// TIA Portal project "GaraznaVrata" (V17)

(* hardware
DEVICE "S7-1200 station_1"  S7-1200 Station
   slot 0: "Rack_0"  S7-1200 Rack  Rack  V1.0
   slot 1: "PLC_1"  CPU 1214C DC/DC/DC  6ES7 214-1AG40-0XB0  V4.2
DEVICE "HMI_1"  TP1200 Comfort
   slot 0: "HMI_1"  TP1200 Comfort  6AV2 124-0MC01-0AX0  17.0.0.0
   slot 1: "HMI_RT_1"  TP1200 Comfort  6AV2 124-0MC01-0AX0  17.0.0.0
   slot 5: "HMI_1.IE_CP_1"  PROFINET Interface  17.0.0.0
      slot 1: "PROFINET Interface_1"  PROFINET Interface
         slot 1: "Port_1"  Port
         slot 2: "Port_2"  Port
   slot 7: "HMI_1.MPI/DP_CP_1"  MPI/DP Interface  17.0.0.0
DEVICE "S7-1500/ET200MP station_1"  S7-1500 station
   slot 0: "Rail_0"  Rack  6ES7 590-1***0-0AA0
   slot 1: "PLC_2"  CPU 1513-1 PN  6ES7 513-1AL01-0AB0  V2.9
      slot 3: "CPU display_1"  6ES7591-1AA00-0AA0
      slot 32768: "PROFINET interface_1"  X1
         slot 32769: "Port_1"  X1 P1
         slot 32770: "Port_2"  X1 P2
      slot 34817: "Virtual CP interface port_1"  Virtual CP interface port  Virtual CP interface port
*)

// ===== PLC "PLC_1"  CPU 1214C DC/DC/DC =====

VAR_GLOBAL   // PLC tag table "Default tag table"
   "System_Byte" AT %MB1 : Byte;
   "FirstScan" AT %M1.0 : Bool;
   "DiagStatusUpdate" AT %M1.1 : Bool;
   "AlwaysTRUE" AT %M1.2 : Bool;
   "AlwaysFALSE" AT %M1.3 : Bool;
   "Clock_Byte" AT %MB0 : Byte;
   "Clock_10Hz" AT %M0.0 : Bool;
   "Clock_5Hz" AT %M0.1 : Bool;
   "Clock_2.5Hz" AT %M0.2 : Bool;
   "Clock_2Hz" AT %M0.3 : Bool;
   "Clock_1.25Hz" AT %M0.4 : Bool;
   "Clock_1Hz" AT %M0.5 : Bool;
   "Clock_0.625Hz" AT %M0.6 : Bool;
   "Clock_0.5Hz" AT %M0.7 : Bool;
END_VAR

VAR_GLOBAL   // PLC tag table "Tag table_1"
   "T1" AT %I0.0 : Bool;
   "T2" AT %I0.1 : Bool;
   "S1" AT %I0.2 : Bool;
   "KO" AT %I0.3 : Bool;
   "KZ" AT %I0.4 : Bool;
   "K1" AT %I0.5 : Bool;
   "K2" AT %I0.6 : Bool;
   "MZS" AT %I0.7 : Bool;
   "OTV" AT %Q0.0 : Bool;
   "ZAT" AT %Q0.1 : Bool;
   "ALM" AT %Q0.2 : Bool;
END_VAR

DATA_BLOCK "Block_2_DB"   // DB2
{ S7_Optimized_Access := 'TRUE' }
VERSION : 0.1
// stored: InstanceOfName Block_2
"Block_2"
BEGIN
END_DATA_BLOCK

FUNCTION_BLOCK "Block_2"   // FB1, SCL
{ S7_Optimized_Access := 'TRUE' }
VERSION : 0.1
   VAR_INPUT
      T1 : Bool;   // Inside push button
      T2 : Bool;   // Outside push button
      S1 : Bool;   // Inside comb switch
      KO : Bool;   // Signal "doors are open"
      KZ : Bool;   // Signal "doors are closed"
      K1 : Bool;   // Doors are opening
      K2 : Bool;   // Doors are closing
      MZS : Bool;   // Motor protection switch
   END_VAR
   VAR_OUTPUT
      OTV : Bool;   // Command to open the door
      ZAT : Bool;   // Command to close the door
      ALM : Bool;   // Alarm
   END_VAR
   VAR_IN_OUT
      M_BIT2 : Bool;   // temp bit for T2
      M_BIT : Bool;   // temp bit for T1
   END_VAR
   VAR
      sAlarm_MZS : Bool;   // Flag for MZS alarm
      sAlarm_KOKZ : Bool;   // Flag for KO and KZ alarm
      sAlarm_stuck : Bool;   // Flag for if gate didnt close/open
      sAlarm_K1K2 : Bool;   // Flag for K1 or K2 alarm
      sCls_gate : Bool;   // Flag to close the door
      sOpn_gate : Bool;   // Flag to open the door
      sGate_dir : Bool;   // Remember the last dirrection of the gate
      sOpening : Bool;   // temp var for opening gate
      sClosing : Bool;   // temp var for closing gate
      IEC_Timer_30s_alarm : TON_TIME;   // Timer for alarm_stuck
      IEC_Timer_5s_alarm : TON_TIME;   // Timer for alarm_K1K2
      IEC_Timer_2min_alarm : TON_TIME;   // Timer when door's are open
   END_VAR
   VAR_TEMP
      xPerm_opn : Bool;   // Permission to open the door
      xPerm_cls : Bool;   // Permission to close the door
      xT : Time;
      xAuto_close : Bool;   // Flag to auto close the door
   END_VAR
   VAR CONSTANT
      timer_2min : Time := T#2m;
      timer_5s : Time := T#5s;
      timer_30s : Time := T#30s;
   END_VAR
BEGIN
     REGION _AUTO_CLOSE
       // If gate is opened more than 2 min close it
       #IEC_Timer_2min_alarm(IN := #KO,
                             PT := #timer_2min,
                             Q => #xAuto_close,
                             ET => #xT);


       IF #xAuto_close THEN
           #sCls_gate := TRUE;
       END_IF;
   END_REGION

     REGION _PERMISSIONS
         // Permissions open the door
         IF #KZ AND NOT (#sAlarm_MZS OR #sAlarm_K1K2 OR #sAlarm_KOKZ OR #sAlarm_stuck) THEN
             #xPerm_opn := TRUE;
         ELSE
             #xPerm_opn := FALSE;
         END_IF;

         // Permission to close the door
         IF #KO AND NOT (#sAlarm_MZS OR #sAlarm_K1K2 OR #sAlarm_KOKZ OR #sAlarm_stuck) THEN
             #xPerm_cls := TRUE;
         ELSE
             #xPerm_cls := FALSE;
         END_IF;
     END_REGION

     REGION _PUSH_BUTTON_EVENT
         // T1 or T2 is pushed
         IF (#T1 AND NOT (#M_BIT)) XOR (#S1 AND (#T2 AND NOT (#M_BIT2))) THEN

             //open
             IF #xPerm_opn THEN
                 #sOpn_gate := TRUE;
             END_IF;

             //close
             IF #xPerm_cls THEN
                 #sCls_gate := TRUE;
             END_IF;

             //resume opening/closing door after error
             IF (#sAlarm_MZS OR #sAlarm_K1K2 OR #sAlarm_KOKZ OR #sAlarm_stuck) = FALSE AND #KO = FALSE AND #KZ = FALSE THEN
                 IF #sGate_dir THEN
                     #sOpn_gate := TRUE;
                 ELSE
                     #sCls_gate := TRUE;
                 END_IF;
             END_IF;

             // alarm shut down
             IF #sAlarm_MZS OR #sAlarm_K1K2 OR #sAlarm_KOKZ OR #sAlarm_stuck THEN
                 #sAlarm_MZS := FALSE;
                 #sAlarm_K1K2 := FALSE;
                 #sAlarm_KOKZ := FALSE;
                 #sAlarm_stuck := FALSE;
             END_IF;

             // set temp variables
             #sOpening := #sOpn_gate;
             #sClosing := #sCls_gate;

         END_IF;

         //set temp bit for edge detecting
         #M_BIT := #T1;
         #M_BIT2 := #T2;
     END_REGION

     REGION _REMEMBER_LAST_DIRRECTION
         // Remember the last direction
         IF #sOpn_gate THEN
             #sGate_dir := TRUE; // last dirrection of the gate was 'open'
         ELSIF #sCls_gate THEN
             #sGate_dir := FALSE; // last dirrection of the gate was 'close'
         END_IF;
     END_REGION

     REGION _OPEN/CLOSE_GATE
         // Start opening
         #OTV := #sOpn_gate;

         // Start Closing
         #ZAT := #sCls_gate;


         // Stop the opening
         IF #KO THEN
             #sOpn_gate := FALSE;
             #sOpening := #sOpn_gate;
         END_IF;

         // Stop the closing
         IF #KZ THEN
             #sCls_gate := FALSE;
             #sClosing := #sCls_gate;
         END_IF;
     END_REGION

     REGION _ALARMS


         (*
           alarm_MZS -> MZS error
           alarm_KOKZ -> Both KZ and K0 are active
           alarm_stuck -> If door didnt close or open within 30sec
           alarm_K1K2 -> Direction confirmation(K1 or K2) did not come within 5 sec of opening/closing gate
          *)

         //Send alarm signal
         IF #sAlarm_MZS OR #sAlarm_K1K2 OR #sAlarm_KOKZ OR #sAlarm_stuck THEN
             #sOpn_gate := FALSE;
             #sCls_gate := FALSE;
             #ALM := "Clock_0.5Hz";
         ELSE
             #ALM := FALSE;
         END_IF;

         //Direction confirmation did not come within 5 sec
         #IEC_Timer_5s_alarm(IN := ((#sOpening AND NOT #K1) OR (#sClosing AND NOT #K2)),
                             PT := #timer_5s,
                             Q => #sAlarm_K1K2,
                             ET => #xT);


         //If door didnt close or open within 30sec
         #IEC_Timer_30s_alarm(IN := #sOpening OR #sClosing,
                              PT := #timer_30s,
                              Q => #sAlarm_stuck,
                              ET => #xT);


         //MZS error
         IF #MZS THEN
             #sAlarm_MZS := TRUE;
         END_IF;

         //Both KZ and K0 are active
         IF #KZ AND #KO THEN
             #sAlarm_KOKZ := TRUE;
         END_IF;

     END_REGION
END_FUNCTION_BLOCK

ORGANIZATION_BLOCK "Main"   // OB1, LAD, ProgramCycle
TITLE = "Main Program Sweep (Cycle)"
{ S7_Optimized_Access := 'TRUE' }
VERSION : 0.1
   VAR_INPUT
      Initial_Call : Bool;   // Initial call of this OB
      Remanence : Bool;   // =True, if remanent data are available
   END_VAR
BEGIN

REGION Network 1
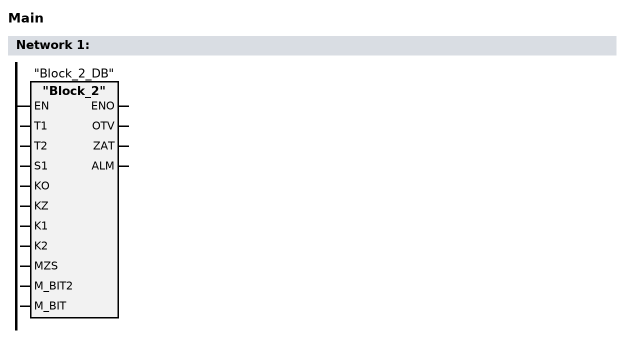
   RUNG wire#powerrail
      "Block_2_DB"(T1 :=, T2 :=, S1 :=, KO :=, KZ :=, K1 :=, K2 :=, MZS :=, OTV =>, ZAT =>, ALM =>, M_BIT :=, M_BIT2 :=)
   END_RUNG
   // the same network as SCL:
   "Block_2_DB"();   // "Block_2"
END_REGION
END_ORGANIZATION_BLOCK

ORGANIZATION_BLOCK "Startup"   // OB100, LAD, Startup
TITLE = "Complete Restart"
{ S7_Optimized_Access := 'TRUE' }
VERSION : 0.1
   VAR_INPUT
      LostRetentive : Bool;   // True if retentive data are lost
      LostRTC : Bool;   // True if date and time are lost
   END_VAR
BEGIN

REGION Network 1
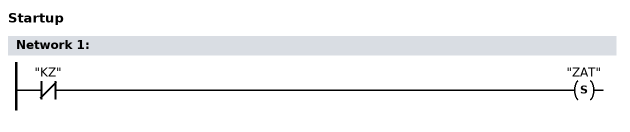
   RUNG wire#powerrail
      I_Contact( "KZ" )
      S_Coil( "ZAT" )
   END_RUNG
   // the same network as SCL:
   IF NOT "KZ" THEN "ZAT" := TRUE; END_IF;
END_REGION
END_ORGANIZATION_BLOCK

// ===== PLC "PLC_2"  CPU 1513-1 PN =====

VAR_GLOBAL   // PLC tag table "Default tag table"
   "ZAT" AT %Q0.1 : Bool;
   "T2" AT %I0.1 : Bool;
   "T1" AT %I0.0 : Bool;
   "System_Byte" AT %MB1 : Byte;
   "S1" AT %I0.2 : Bool;
   "OTV" AT %Q0.0 : Bool;
   "MZS" AT %I0.7 : Bool;
   "KZ" AT %I0.4 : Bool;
   "KO" AT %I0.3 : Bool;
   "K2" AT %I0.6 : Bool;
   "K1" AT %I0.5 : Bool;
   "FirstScan" AT %M1.0 : Bool;
   "DiagStatusUpdate" AT %M1.1 : Bool;
   "Clock_Byte" AT %MB0 : Byte;
   "Clock_5Hz" AT %M0.1 : Bool;
   "Clock_2Hz" AT %M0.3 : Bool;
   "Clock_2.5Hz" AT %M0.2 : Bool;
   "Clock_1Hz" AT %M0.5 : Bool;
   "Clock_10Hz" AT %M0.0 : Bool;
   "Clock_1.25Hz" AT %M0.4 : Bool;
   "Clock_0.625Hz" AT %M0.6 : Bool;
   "Clock_0.5Hz" AT %M0.7 : Bool;
   "AlwaysTRUE" AT %M1.2 : Bool;
   "AlwaysFALSE" AT %M1.3 : Bool;
   "ALM" AT %Q0.2 : Bool;
END_VAR

DATA_BLOCK "Block_2_DB"   // DB2
{ S7_Optimized_Access := 'TRUE' }
VERSION : 0.1
// stored: InstanceOfName Block_2
"Block_2"
BEGIN
END_DATA_BLOCK

FUNCTION_BLOCK "Block_2"   // FB1, SCL
{ S7_Optimized_Access := 'TRUE' }
VERSION : 0.1
   VAR_INPUT
      T1 : Bool;   // Inside push button
      T2 : Bool;   // Outside push button
      S1 : Bool;   // Inside comb switch
      KO : Bool;   // Signal "doors are open"
      KZ : Bool;   // Signal "doors are closed"
      K1 : Bool;   // Doors are opening
      K2 : Bool;   // Doors are closing
      MZS : Bool;   // Motor protection switch
   END_VAR
   VAR_OUTPUT
      OTV : Bool;   // Command to open the door
      ZAT : Bool;   // Command to close the door
      ALM : Bool;   // Alarm
   END_VAR
   VAR_IN_OUT
      M_BIT2 : Bool;   // temp bit for T2
      M_BIT : Bool;   // temp bit for T1
   END_VAR
   VAR
      sAlarm_MZS : Bool;   // Flag for MZS alarm
      sAlarm_KOKZ : Bool;   // Flag for KO and KZ alarm
      sAlarm_stuck : Bool;   // Flag for if gate didnt close/open
      sAlarm_K1K2 : Bool;   // Flag for K1 or K2 alarm
      sCls_gate : Bool;   // Flag to close the door
      sOpn_gate : Bool;   // Flag to open the door
      sGate_dir : Bool;   // Remember the last dirrection of the gate
      sOpening : Bool;   // temp var for opening gate
      sClosing : Bool;   // temp var for closing gate
      IEC_Timer_30s_alarm : TON_TIME;   // Timer for alarm_stuck
      IEC_Timer_5s_alarm : TON_TIME;   // Timer for alarm_K1K2
      IEC_Timer_2min_alarm : TON_TIME;   // Timer when door's are open
   END_VAR
   VAR_TEMP
      xPerm_opn : Bool;   // Permission to open the door
      xPerm_cls : Bool;   // Permission to close the door
      xT : Time;
      xAuto_close : Bool;   // Flag to auto close the door
   END_VAR
   VAR CONSTANT
      timer_2min : Time := T#2m;
      timer_5s : Time := T#5s;
      timer_30s : Time := T#30s;
   END_VAR
BEGIN
     REGION _AUTO_CLOSE
       // If gate is opened more than 2 min close it
       #IEC_Timer_2min_alarm(IN := #KO,
                             PT := #timer_2min,
                             Q => #xAuto_close,
                             ET => #xT);


       IF #xAuto_close THEN
           #sCls_gate := TRUE;
       END_IF;
   END_REGION

     REGION _PERMISSIONS
         // Permissions open the door
         IF #KZ AND NOT (#sAlarm_MZS OR #sAlarm_K1K2 OR #sAlarm_KOKZ OR #sAlarm_stuck) THEN
             #xPerm_opn := TRUE;
         ELSE
             #xPerm_opn := FALSE;
         END_IF;

         // Permission to close the door
         IF #KO AND NOT (#sAlarm_MZS OR #sAlarm_K1K2 OR #sAlarm_KOKZ OR #sAlarm_stuck) THEN
             #xPerm_cls := TRUE;
         ELSE
             #xPerm_cls := FALSE;
         END_IF;
     END_REGION

     REGION _PUSH_BUTTON_EVENT
         // T1 or T2 is pushed
         IF (#T1 AND NOT (#M_BIT)) XOR (#S1 AND (#T2 AND NOT (#M_BIT2))) THEN

             //open
             IF #xPerm_opn THEN
                 #sOpn_gate := TRUE;
             END_IF;

             //close
             IF #xPerm_cls THEN
                 #sCls_gate := TRUE;
             END_IF;

             //resume opening/closing door after error
             IF (#sAlarm_MZS OR #sAlarm_K1K2 OR #sAlarm_KOKZ OR #sAlarm_stuck) = FALSE AND #KO = FALSE AND #KZ = FALSE THEN
                 IF #sGate_dir THEN
                     #sOpn_gate := TRUE;
                 ELSE
                     #sCls_gate := TRUE;
                 END_IF;
             END_IF;

             // alarm shut down
             IF #sAlarm_MZS OR #sAlarm_K1K2 OR #sAlarm_KOKZ OR #sAlarm_stuck THEN
                 #sAlarm_MZS := FALSE;
                 #sAlarm_K1K2 := FALSE;
                 #sAlarm_KOKZ := FALSE;
                 #sAlarm_stuck := FALSE;
             END_IF;

             // set temp variables
             #sOpening := #sOpn_gate;
             #sClosing := #sCls_gate;

             #T1 := FALSE;
             #T2 := FAlSE;

         END_IF;

         //set temp bit for edge detecting
         #M_BIT := #T1;
         #M_BIT2 := #T2;
     END_REGION

     REGION _REMEMBER_LAST_DIRRECTION
         // Remember the last direction
         IF #sOpn_gate THEN
             #sGate_dir := TRUE; // last dirrection of the gate was 'open'
         ELSIF #sCls_gate THEN
             #sGate_dir := FALSE; // last dirrection of the gate was 'close'
         END_IF;
     END_REGION

     REGION _OPEN/CLOSE_GATE
         // Start opening
         #OTV := #sOpn_gate;

         // Start Closing
         #ZAT := #sCls_gate;


         // Stop the opening
         IF #KO THEN
             #sOpn_gate := FALSE;
             #sOpening := #sOpn_gate;
         END_IF;

         // Stop the closing
         IF #KZ THEN
             #sCls_gate := FALSE;
             #sClosing := #sCls_gate;
         END_IF;
     END_REGION

     REGION _ALARMS


         (*
           alarm_MZS -> MZS error
           alarm_KOKZ -> Both KZ and K0 are active
           alarm_stuck -> If door didnt close or open within 30sec
           alarm_K1K2 -> Direction confirmation(K1 or K2) did not come within 5 sec of opening/closing gate
          *)

         //Send alarm signal
         IF #sAlarm_MZS OR #sAlarm_K1K2 OR #sAlarm_KOKZ OR #sAlarm_stuck THEN
             #sOpn_gate := FALSE;
             #sCls_gate := FALSE;
             #ALM := "Clock_0.5Hz";
         ELSE
             #ALM := FALSE;
         END_IF;

         //Direction confirmation did not come within 5 sec
         #IEC_Timer_5s_alarm(IN := ((#sOpening AND NOT #K1) OR (#sClosing AND NOT #K2)),
                             PT := #timer_5s,
                             Q => #sAlarm_K1K2,
                             ET => #xT);


         //If door didnt close or open within 30sec
         #IEC_Timer_30s_alarm(IN := #sOpening OR #sClosing,
                              PT := #timer_30s,
                              Q => #sAlarm_stuck,
                              ET => #xT);


         //MZS error
         IF #MZS THEN
             #sAlarm_MZS := TRUE;
         END_IF;

         //Both KZ and K0 are active
         IF #KZ AND #KO THEN
             #sAlarm_KOKZ := TRUE;
         END_IF;

     END_REGION
END_FUNCTION_BLOCK

ORGANIZATION_BLOCK "Main"   // OB1, LAD, ProgramCycle
TITLE = "Main Program Sweep (Cycle)"
{ S7_Optimized_Access := 'TRUE' }
VERSION : 0.1
   VAR_INPUT
      Initial_Call : Bool;   // Initial call of this OB
      Remanence : Bool;   // =True, if remanent data are available
   END_VAR
   VAR_TEMP
      ok : Int;
   END_VAR
BEGIN

REGION Network 1: WWW DB
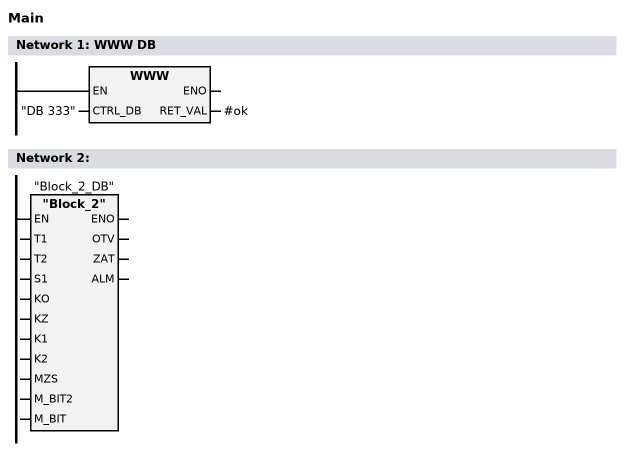
   #ok := WWW(CTRL_DB := "DB 333");
END_REGION

REGION Network 2
   RUNG wire#powerrail
      "Block_2_DB"(T1 :=, T2 :=, S1 :=, KO :=, KZ :=, K1 :=, K2 :=, MZS :=, OTV =>, ZAT =>, ALM =>, M_BIT :=, M_BIT2 :=)
   END_RUNG
   // the same network as SCL:
   "Block_2_DB"();   // "Block_2"
END_REGION
END_ORGANIZATION_BLOCK

ORGANIZATION_BLOCK "Startup"   // OB100, LAD, Startup
TITLE = "Complete Restart"
{ S7_Optimized_Access := 'TRUE' }
VERSION : 0.1
   VAR_INPUT
      LostRetentive : Bool;   // True if retentive data are lost
      LostRTC : Bool;   // True if date and time are lost
   END_VAR
BEGIN

REGION Network 1: Command to close the door
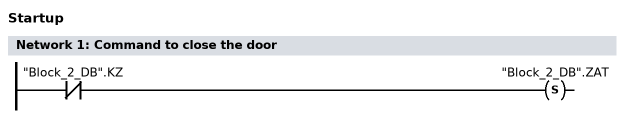
   RUNG wire#powerrail
      I_Contact( "Block_2_DB".KZ )
      S_Coil( "Block_2_DB".ZAT )
   END_RUNG
   // the same network as SCL:
   IF NOT "Block_2_DB".KZ THEN "Block_2_DB".ZAT := TRUE; END_IF;
END_REGION
END_ORGANIZATION_BLOCK

(* ===== HMI "HMI_RT_1" =====
system functions are stored by id; their names below are inferred from use
connection "HMI_Connection_1": ETHERNET, S7_1200_OMS
connection "HMI_Connection_2": ETHERNET, S7_1500_OMS

HMI tags "Default tag table"
   "Tag_ScreenNumber" : UInt, internal
   "Block_2_DB_T1" : Bool = PLC Block_2_DB.T1, 1 s
   "Block_2_DB_T2" : Bool = PLC Block_2_DB.T2, 1 s
   "Block_2_DB_S1" : Bool = PLC Block_2_DB.S1, 1 s
   "Block_2_DB_KZ" : Bool = PLC Block_2_DB.KZ, 1 s
   "Block_2_DB_KO" : Bool = PLC Block_2_DB.KO, 1 s
   "Block_2_DB_K1" : Bool = PLC Block_2_DB.K1, 1 s
   "Block_2_DB_K2" : Bool = PLC Block_2_DB.K2, 1 s
   "Block_2_DB_MZS" : Bool = PLC Block_2_DB.MZS, 1 s
   "Block_2_DB_OTV" : Bool = PLC Block_2_DB.OTV, 1 s
   "Block_2_DB_ZAT" : Bool = PLC Block_2_DB.ZAT, 1 s
   "Block_2_DB_ALM" : Bool = PLC Block_2_DB.ALM AT %DB1.DBX0.0, 1 s

screen "Root screen" 1280x740, template "Template_1"
   TextField "HmiScreenItemData_1" at 89,3 size 1024x27; Text 'Welcome to my garage door's'
   Button "HmiScreenItemData" at 36,36 size 159x47; TextOff 'Screen0'; PictureOff "Navigates to Screen0 for TP1200 Comfort 17.0.0.0"; PictureOn "Navigates to Screen0 for TP1200 Comfort 17.0.0.0"
      on Release: ActivateScreen("Screen0", 0)
   Button "HmiScreenItemData_2" at 36,95 size 159x47; TextOff 'System screens'; PictureOff "Navigates to System screens for TP1200 Comfort 17.0.0.0"; PictureOn "Navigates to System screens for TP1200 Comfort 17.0.0.0"
      on Release: ActivateScreen("System screens", 0)
   Button "Button_1" at 37,158 size 157x47; TextOff 'T1'
      on Press: function_b14e0dd5("Block_2_DB_T1", 0)
      Appearance <- "Block_2_DB_T1"
   Button "Button_2" at 38,308 size 157x47; TextOff 'T2'
      on Press: function_b14e0dd5("Block_2_DB_T2", 0)
      Appearance <- "Block_2_DB_T2"
   Switch "Switch_1" at 48,215 size 136x69; CaptionText 'S1'; TextOff 'OFF'; TextOn 'ON'
      ProcessValue <- "Block_2_DB_S1"
   Button "Button_3" at 37,386 size 157x47; TextOff 'KO'
      Appearance <- "Block_2_DB_KO"
      on Click: InvertBit("Block_2_DB_KO")
   Button "Button_4" at 37,446 size 157x47; TextOff 'KZ'
      Appearance <- "Block_2_DB_KZ"
      on Press: InvertBit("Block_2_DB_KZ")
   Button "Button_5" at 36,506 size 157x47; TextOff 'K1'
      on Click: InvertBit("Block_2_DB_K1")
      Appearance <- "Block_2_DB_K1"
   Button "Button_6" at 37,563 size 157x47; TextOff 'K2'
      on Click: InvertBit("Block_2_DB_K2")
      Appearance <- "Block_2_DB_K2"
   Button "Button_10" at 37,622 size 157x47; TextOff 'MZS'
      Appearance <- "Block_2_DB_MZS"
      on Press: function_b14e0dd5("Block_2_DB_MZS", 0)
   Circle "Circle_1" at 966,185 size 38x38
      Appearance <- "Block_2_DB_OTV"
   TextField "Text field_1" at 1029,189 size 201x28; Text 'Garage doors opening'
   Circle "Circle_2" at 966,365 size 38x38
      Appearance <- "Block_2_DB_KZ"
   TextField "Text field_2" at 1028,369 size 210x28; Text 'Garage doors are close'
   Circle "Circle_3" at 966,458 size 38x38
      Appearance <- "Block_2_DB_ALM"
   TextField "Text field_3" at 1029,462 size 48x28; Text 'Error'
      Appearance <- "Block_2_DB_ALM"
   Circle "Circle_4" at 966,234 size 38x38
      Appearance <- "Block_2_DB_KO"
   TextField "Text field_4" at 1029,238 size 209x28; Text 'Garage doors are open'
   Circle "Circle_5" at 966,313 size 38x38
      Appearance <- "Block_2_DB_ZAT"
   TextField "Text field_5" at 1029,317 size 191x28; Text 'Garage doors closing'
   Rectangle "Rectangle_3" at 348,176 size 497x448
      Visibility <- "Block_2_DB_KO"
   Rectangle "Rectangle_4" at 348,176 size 497x449
      Visibility <- "Block_2_DB_KZ"

Template "Template_1" 1280x740
   Button "Exit" at 1200,679 size 78x59; TextOff 'Exit'; PictureOff "ExitRuntime_TP1200_Comfort_TR"; PictureOn "ExitRuntime_TP1200_Comfort_TR"
      on Release: StopRuntime(0)
   Button "Log on" at 1120,679 size 78x59; TextOff 'Log on'; PictureOff "Login_TP1200_Comfort_TR"; PictureOn "Login_TP1200_Comfort_TR"
      on Release: function_a2a04561()
   Button "Language" at 1040,679 size 78x59; TextOff 'Language'; PictureOff "ToggleLanguage_TP1200_Comfort_TR"; PictureOn "ToggleLanguage_TP1200_Comfort_TR"
      on Release: function_fb9197e8(-1)
   Button "Template_Button" at 960,679 size 78x59; TextOff 'Text'
   Button "Template_Button_1" at 880,679 size 78x59; TextOff 'Text'
   Button "Template_Button_2" at 800,679 size 78x59; TextOff 'Text'
   Button "Template_Button_3" at 720,679 size 78x59; TextOff 'Text'
   Button "Template_Button_4" at 640,679 size 78x59; TextOff 'Text'
   Button "Template_Button_5" at 561,679 size 78x59; TextOff 'Text'
   Button "Template_Button_6" at 481,679 size 78x59; TextOff 'Text'
   Button "Template_Button_7" at 401,679 size 78x59; TextOff 'Text'
   Button "Template_Button_8" at 321,679 size 78x59; TextOff 'Text'
   Button "Template_Button_9" at 241,679 size 78x59; TextOff 'Text'
   Button "Template_Button_10" at 161,679 size 78x59; TextOff 'Text'
   Button "Alarms" at 81,679 size 78x59; TextOff 'Alarms'; PictureOff "AlarmDisplay_TP1200_Comfort_TR"; PictureOn "AlarmDisplay_TP1200_Comfort_TR"
      on Release: function_ef3f5d25("Alarm window_Unacknowledged", -1)
   Button "Start screen" at 1,679 size 78x59; TextOff 'Start screen'; PictureOff "NavigateHome_TP1200_Comfort_TR"; PictureOn "NavigateHome_TP1200_Comfort_TR"
      on Release: ActivateScreen("Root screen", 0)

screen "Screen0" 1280x740, template "Template_1"
   on GenerateScreen: SetTag("Tag_ScreenNumber", 2)
   TextField "HmiScreenItemData" at 128,324 size 1024x27; Text 'Screen0'
   Button "Back" at 1,1 size 159x47; TextOff 'Back'
      on Release: ActivateScreen("Root screen", 0)
   Button "HmiScreenItemData_1" at 36,95 size 159x47; TextOff 'Screen1'; PictureOff "Navigates to Screen1 for TP1200 Comfort 17.0.0.0"; PictureOn "Navigates to Screen1 for TP1200 Comfort 17.0.0.0"
      on Release: ActivateScreen("Screen1", 0)

screen "Screen1" 1280x740, template "Template_1"
   on GenerateScreen: SetTag("Tag_ScreenNumber", 3)
   TextField "HmiScreenItemData" at 128,324 size 1024x27; Text 'Screen1'
   Button "Back" at 1,1 size 159x47; TextOff 'Back'
      on Release: ActivateScreen("Screen0", 0)

screen "System screens" 1280x740, template "Template_1"
   on GenerateScreen: SetTag("Tag_ScreenNumber", 4)
   Button "Back" at 1,1 size 159x47; TextOff 'Back'
      on Release: ActivateScreen("Root screen", 0)
   Button "HmiScreenItemData" at 36,95 size 159x47; TextOff 'SIMATIC PLC system diagnos...'; PictureOff "Navigates to SIMATIC PLC system diagnostics for TP1200 Comfort 17.0.0.0"; PictureOn "Navigates to SIMATIC PLC system diagnostics for TP1200 Comfort 17.0.0.0"
      on Release: ActivateScreen("SIMATIC PLC system diagnostics", 0)
   Button "HmiScreenItemData_1" at 36,154 size 159x47; TextOff 'Project information'; PictureOff "Navigates to Project information for TP1200 Comfort 17.0.0.0"; PictureOn "Navigates to Project information for TP1200 Comfort 17.0.0.0"
      on Release: ActivateScreen("Project information", 0)
   Button "HmiScreenItemData_2" at 36,213 size 159x47; TextOff 'System settings'; PictureOff "Navigates to System settings for TP1200 Comfort 17.0.0.0"; PictureOn "Navigates to System settings for TP1200 Comfort 17.0.0.0"
      on Release: ActivateScreen("System settings", 0)
   Button "HmiScreenItemData_3" at 36,272 size 159x47; TextOff 'User administration'; PictureOff "Navigates to User administration for TP1200 Comfort 17.0.0.0"; PictureOn "Navigates to User administration for TP1200 Comfort 17.0.0.0"
      on Release: ActivateScreen("User administration", 0)
   Button "HmiScreenItemData_4" at 36,331 size 159x47; TextOff 'System information'; PictureOff "Navigates to System information for TP1200 Comfort 17.0.0.0"; PictureOn "Navigates to System information for TP1200 Comfort 17.0.0.0"
      on Release: ActivateScreen("System information", 0)
   Button "HmiScreenItemData_5" at 36,390 size 159x47; TextOff 'Different jobs'; PictureOff "Navigates to Different jobs for TP1200 Comfort 17.0.0.0"; PictureOn "Navigates to Different jobs for TP1200 Comfort 17.0.0.0"
      on Release: ActivateScreen("Different jobs", 0)

screen "SIMATIC PLC system diagnostics" 1280x740, template "Template_1"
   on GenerateScreen: SetTag("Tag_ScreenNumber", 5)
   SysDiagControl "HmiScreenItemData" at 1,49 size 1276x623
   Button "Back" at 1,1 size 159x47; TextOff 'Back'
      on Release: ActivateScreen("System screens", 0)

screen "Project information" 1280x740, template "Template_1"
   on GenerateScreen: SetTag("Tag_ScreenNumber", 6)
   TextField "HmiScreenItemData" at 35,51 size 171x28; Text 'Project name:'
   TextField "HmiScreenItemData_1" at 241,51 size 1004x28; Text 'GaraznaVrata'
   TextField "HmiScreenItemData_2" at 35,81 size 171x28; Text 'Created on:'
   TextField "HmiScreenItemData_3" at 241,81 size 1004x28; Text '10/8/2021 2:57:25 PM'
   TextField "HmiScreenItemData_4" at 35,111 size 171x28; Text 'Author:'
   TextField "HmiScreenItemData_5" at 241,111 size 1004x28; Text 'atomgmt'
   TextField "HmiScreenItemData_6" at 35,141 size 171x28; Text 'Description:'
   TextField "HmiScreenItemData_7" at 241,141 size 1004x28; Text 'This panel was made as a part of internship program to test the 'garage door' assignment'
   Button "Back" at 1,1 size 159x47; TextOff 'Back'
      on Release: ActivateScreen("System screens", 0)

screen "System settings" 1280x740, template "Template_1"
   on GenerateScreen: SetTag("Tag_ScreenNumber", 7)
   Button "Calibrate screen" at 36,95 size 159x47; TextOff 'Calibrate screen'
      on Release: function_bc3e350c()
   Button "Clean screen" at 36,154 size 159x47; TextOff 'Clean screen'
      on Release: function_be740847(30)
   Button "Back" at 1,1 size 159x47; TextOff 'Back'
      on Release: ActivateScreen("System screens", 0)

screen "User administration" 1280x740, template "Template_1"
   on GenerateScreen: SetTag("Tag_ScreenNumber", 8)
   UserView "HmiScreenItemData" at 1,49 size 1276x623
   Button "Back" at 1,1 size 159x47; TextOff 'Back'
      on Release: ActivateScreen("System screens", 0)

screen "System information" 1280x740, template "Template_1"
   on GenerateScreen: SetTag("Tag_ScreenNumber", 9)
   TextField "HmiScreenItemData" at 35,51 size 171x28; Text 'HMI device type:'
   TextField "HmiScreenItemData_1" at 241,51 size 1004x28; Text 'TP1200 Comfort 17.0.0.0'
   TextField "HmiScreenItemData_2" at 35,81 size 171x28; Text 'Version:'
   TextField "HmiScreenItemData_3" at 35,111 size 171x28; Text 'Connection:'
   TextField "HmiScreenItemData_4" at 241,111 size 1004x28; Text 'ETHERNET'
   TextField "HmiScreenItemData_5" at 35,141 size 171x28; Text 'PLC:'
   TextField "HmiScreenItemData_6" at 241,141 size 1004x28; Text 'SIMATIC S7 1200'
   Button "Display version" at 241,81 size 1004x28; TextOff 'Display version'
      on Release: function_febcb963(-1)
   Button "Back" at 1,1 size 159x47; TextOff 'Back'
      on Release: ActivateScreen("System screens", 0)

screen "Different jobs" 1280x740, template "Template_1"
   on GenerateScreen: SetTag("Tag_ScreenNumber", 10)
   Button "Online" at 36,95 size 159x47; TextOff 'Online'
      on Release: function_bb44b551(0)
   Button "Offline" at 36,154 size 159x47; TextOff 'Offline'
      on Release: function_bb44b551(1)
   Button "Transfer" at 36,213 size 159x47; TextOff 'Transfer'
      on Release: function_bb44b551(2)
   Button "Toggle language" at 36,272 size 159x47; TextOff 'Toggle language'
      on Release: function_fb9197e8(-1)
   Button "Control Panel" at 36,331 size 159x47; TextOff 'Control Panel'
      on Release: function_f34a74f3()
   Button "Stop Runtime" at 36,390 size 159x47; TextOff 'Stop Runtime'
      on Release: StopRuntime(0)
   Button "Back" at 1,1 size 159x47; TextOff 'Back'
      on Release: ActivateScreen("System screens", 0)
*)